FUNCTION "LGF_MergeBytesToDWord" : DWord
TITLE = LGF_MergeBytesToDWord
{ S7_Optimized_Access := 'TRUE' }
AUTHOR : Siemens_Digital_Industry
FAMILY : LGF
NAME : LGF_MergeBytesToDWord
//This function merge 4 Byte variables into one DWord variable.
   VAR_INPUT
      byte3 : Byte;   // Input Byte 3 - MSB
      byte2 : Byte;   // Input Byte 2
      byte1 : Byte;   // Input Byte 1
      byte0 : Byte;   // Input Byte 0 - LSB
   END_VAR

   VAR_TEMP
      tempDWord : DWord;   // Temp memory to merge Bytes into a DWord
   END_VAR


BEGIN
	REGION BLOCK INFO HEADER
	  //===============================================================================
	  // SIEMENS AG / (c)Copyright 2018
	  //-------------------------------------------------------------------------------
	  // Title:            LGF_MergeBytesToDWord
	  // Comment/Function: This function merge 4 Byte variables into one DWord variable.
	  // Library/Family:   LGF (Library General Functions)
	  // Author:           Siemens Digital Industry Support
	  // Tested with:      S7-PLCSIM Advanced V2.0 SP1
	  // Engineering:      TIA Portal V14 / V14SP1
	  // Restrictions:     ENO disabled - no error handling, no failure possible.
	  // Requirements:     PLC (S7-1200 / S7-1500)
	  //-------------------------------------------------------------------------------
	  // Change log table:
	  // Version  | Date       | Expert in charge       | Changes applied
	  //----------|------------|------------------------|------------------------------
	  // 01.00.00 | 20.06.2019 | Simatic Systems Support
	  //                         First release
	  // 03.00.00 | 23.04.2020 | Simatic Systems Support | Set version to V3.0.0
	  //                         harmonize the version of the whole library
	  // 03.00.01 | 22.02.2021 | Simatic Systems Support
	  //                         Insert documentation
	  //=============================================================================
	END_REGION

	REGION MERGE
	  // set the bytes by slice access
	  #tempDWord.%B3 := #byte3;
	  #tempDWord.%B2 := #byte2;
	  #tempDWord.%B1 := #byte1;
	  #tempDWord.%B0 := #byte0;
	END_REGION

	REGION OUTPUT
	  #LGF_MergeBytesToDWord := #tempDWord;
	  // no error handling needed
	  ENO := TRUE;
	END_REGION

END_FUNCTION

